(* CoDeSys 2.3.9.50 project: BallGame_template_with_PackMLandDriveFB.pro *)
(* Libraries: TcBase.lib 14.5.09 12:14:08, TcSystem.lib 7.6.16 11:01:22, STANDARD.LIB 5.6.98 12:03:02 *)

(* Task configuration *)
TASK BallGame (PRIORITY := 1, INTERVAL := T#10ms);
	PRG_HMI();
	MAIN();
END_TASK
TASK Drive (PRIORITY := 0, INTERVAL := T#5ms);
	PRG_Drive_Link();
END_TASK

(* Global variable list: Global_Variables *)
VAR_GLOBAL
(* -------------INPUTS and OUTPUTS -------------------*)
(* See Global_Variables_TwinCAT and Global_Variables_CodeSys for
environment specific physical IOs *)

(*-----------------------TIMERS----------------------------*)
	TONMove_Ball_Delay	: TON;
	TONDrive_Delay		: TON;

(*-----------------------COUNTERS----------------------------*)
	CountBallsSortedMetal			: INT:=0;	(*Balls sorted: Metal*)
	CountBallsSortedWooden		: INT:=0;	(*Balls sorted: Wood*)
	CountBallsSortedYellow		: INT:=0;	(*Balls sorted: Wood, Yellow*)
	CountBallsSortedRed			: INT:=0;	(*Balls sorted: Wood, Red*)
	CountBallsSortedBlue			: INT:=0;	(*Balls sorted: Wood, Blue*)
	CountBallsSortedGarbage		: INT:=0;	(*Balls sorted: Unknown*)
	arrCountBallsOnTubes	: ARRAY [1..4] OF INT;	(*Balls on tubes: 1=lower, 2=middle, 3=upper, 4=garbage*)

(*-----------------------FUNCTION BLOCKS----------------*)
	fbDrive				: FB_DriveMovement2;		(*FB for executing the motion*)
	fbStateModel			: FB_StateModel_ST;		(*FB for executing state model*)

(* -------------HMI INPUTS (from HMI to PLC) -------------------*)
	bHMI_BtnStart		: BOOL;		(*Start button on HMI*)

(* -------------HMI OUTPUTS (from PLC to HMI) -------------------*)
	PLC_uModeCurrent	: UINT;		(*Current Mode*)
	PLC_uStateCurrent	: UINT;		(*Current State*)
	O_Light_BeaconRed	: BOOL;		(*Light beacon: Red*)

(*-----------------------OTHER GLOBAL VARS ----------------*)


END_VAR

VAR_GLOBAL CONSTANT
(*-----------------------Lift Position Constants----------------------------*)
	GPOS_LOADING		: WORD := 16#0A;	(*Drive to loading level*)
	GPOS_PIPE_LOW	: WORD := 16#0B;	(*Drive to lower pipe*)
	GPOS_PIPE_MID		: WORD := 16#0C;	(*Drive to middle pipe*)
	GPOS_PIPE_UP		: WORD := 16#0D;	(*Drive to upper pipe*)
	GPOS_GARBAGE		: WORD := 16#0E;	(*Drive to garbage pipe*)
	GPOS_COLOR_SEN	: WORD := 16#0F;	(*Drive to colour sensor*)

(*-----------------------Ball Type Constants----------------------------*)
	METAL				: BOOL := FALSE;
	WOODEN		: BOOL := TRUE;

(*-----------------------TIME Constants----------------------------*)
	T_LOADING_BALL	: TIME := T#1.5s;	(*Delay for ball to roll from Slot2 to Lifter*)
	T_DRIVE_DELAY		: TIME := T#2s;	(*Delay for drive to start movement*)
END_VAR

(* Global variable list: Global_Variables_CodeSys *)
VAR_GLOBAL
(* -------------INPUTS-------------------*)
	ISensorOpt 			:BOOL;	(*Optical sensor - is ball present*)
	ISensorInd 			:BOOL;	(*Inductive sensor - is metal ball present*)
	IEmergencyClear 		:BOOL;	(*Emergency stop is cleared*)
	IRun 				:BOOL;	(*Run switch*)
	ILimitUp 				:BOOL;	(*Lift's limit switch is activated - Up*)
	ILimitLow 		 	:BOOL;	(*Lift's limit switch is activated - Low*)
	IGateClosedMid		:BOOL;	(*Pipe gate closed - Mid*)
	IGateClosedLow		:BOOL;	(*Pipe gate closed - Low*)
	ISorterGateClosed		:BOOL;	(*Sorter gate closed*)
	ISorterLiftUp			:BOOL;	(*Sorter lift at up position*)
	ISorterLiftDown		:BOOL;	(*Sorter lift at down position*)
	IPressureApplied		:BOOL;	(*Pressure is available for the system*)
	TEMP1				:BOOL;
	ISenColourYellow		:BOOL;	(*Colour sensor In1 - Yellow*)
	ISenColourBlue		:BOOL;	(*Colour sensor In2 - Blue*)
	ISenColourGreen		:BOOL;	(*Colour sensor In3 - Green*)
	ISenColourRed		:BOOL;	(*Colour sensor In4 - Red*)
	IDriveStatus 			:WORD;	(*From lift drive status information*)

(* -------------OUTPUTS-------------------*)
	OGateMid			:BOOL;	(*Valve: Open pipe gate - Mid*)
	OGateLow			:BOOL;	(*Valve: Open pipe gate - Low*)
	OSorterGate			:BOOL;	(*Valve: Open sorter gate*)
	OSorterLift			:BOOL;	(*Valve: Sorter lift up*)
	OEjector				:BOOL;	(*Ejector push ball out from lift*)
	ODriveControl 		:WORD;	(*To lift drive control information*)
END_VAR

(* Global variable list: Global_Variables_TwinCAT *)
VAR_GLOBAL
(* -------------INPUTS-------------------*)
	ISensorOpt 		AT %I*	:BOOL;	(*Optical sensor - is ball present*)
	ISensorInd 		AT %I*	:BOOL;	(*Inductive sensor - is metal ball present*)
	IEmergencyClear 	AT %I*	:BOOL;	(*Emergency stop is cleared*)
	IRun 			AT %I*	:BOOL;	(*Run switch*)
	ILimitUp 			AT %I*	:BOOL;	(*Lift's limit switch is activated - Up*)
	ILimitLow 		AT %I* 	:BOOL;	(*Lift's limit switch is activated - Low*)
	IGateClosedMid	AT %I*	:BOOL;	(*Pipe gate closed - Mid*)
	IGateClosedLow	AT %I*	:BOOL;	(*Pipe gate closed - Low*)
	ISorterGateClosed	AT %I*	:BOOL;	(*Sorter gate closed*)
	ISorterLiftUp		AT %I*	:BOOL;	(*Sorter lift at up position*)
	ISorterLiftDown	AT %I*	:BOOL;	(*Sorter lift at down position*)
	IPressureApplied	AT %I*	:BOOL;	(*Pressure is available for the system*)
	TEMP1			AT %I*	:BOOL;
	ISenColourYellow	AT %I*	:BOOL;	(*Colour sensor In1 - Yellow*)
	ISenColourBlue	AT %I*	:BOOL;	(*Colour sensor In2 - Blue*)
	ISenColourGreen	AT %I*	:BOOL;	(*Colour sensor In3 - Green*)
	ISenColourRed	AT %I*	:BOOL;	(*Colour sensor In4 - Red*)
	IDriveStatus 		AT %I*	:WORD;	(*From lift drive status information*)

(* -------------OUTPUTS-------------------*)
	OGateMid		AT %Q*	:BOOL;	(*Valve: Open pipe gate - Mid*)
	OGateLow		AT %Q*	:BOOL;	(*Valve: Open pipe gate - Low*)
	OSorterGate		AT %Q*	:BOOL;	(*Valve: Open sorter gate*)
	OSorterLift		AT %Q*	:BOOL;	(*Valve: Sorter lift up*)
	OEjector			AT %Q*	:BOOL;	(*Ejector push ball out from lift*)
	ODriveControl 	AT %Q*	:WORD;	(*To lift drive control information*)
END_VAR

(* Global variable list: TwinCAT_Configuration *)
(* Generated automatically by TwinCAT - (read only) *)
VAR_CONFIG
	.ISensorOpt AT %IX0.0 : BOOL;	(*  ~ {LinkedWith:TIID^Device 4 (EL6731)^Box 2  (BK3110)^Term 2 (KL1002)^Channel 1^Input} *)
	.ISensorInd AT %IX0.1 : BOOL;	(*  ~ {LinkedWith:TIID^Device 4 (EL6731)^Box 2  (BK3110)^Term 2 (KL1002)^Channel 2^Input} *)
	.IEmergencyClear AT %IX0.2 : BOOL;	(*  ~ {LinkedWith:TIID^Device 4 (EL6731)^Box 2  (BK3110)^Term 3 (KL1002)^Channel 1^Input} *)
	.IRun AT %IX0.3 : BOOL;	(*  ~ {LinkedWith:TIID^Device 4 (EL6731)^Box 2  (BK3110)^Term 3 (KL1002)^Channel 2^Input} *)
	.ILimitUp AT %IX0.4 : BOOL;	(*  ~ {LinkedWith:TIID^Device 4 (EL6731)^Box 2  (BK3110)^Term 4 (KL1002)^Channel 1^Input} *)
	.ILimitLow AT %IX0.5 : BOOL;	(*  ~ {LinkedWith:TIID^Device 4 (EL6731)^Box 2  (BK3110)^Term 4 (KL1002)^Channel 2^Input} *)
	.IGateClosedMid AT %IX0.7 : BOOL;	(*  ~ {LinkedWith:TIID^Device 4 (EL6731)^Box 2  (BK3110)^Term 5 (KL1104)^Channel 2^Input} *)
	.IGateClosedLow AT %IX1.0 : BOOL;	(*  ~ {LinkedWith:TIID^Device 4 (EL6731)^Box 2  (BK3110)^Term 5 (KL1104)^Channel 3^Input} *)
	.ISorterGateClosed AT %IX1.1 : BOOL;	(*  ~ {LinkedWith:TIID^Device 4 (EL6731)^Box 2  (BK3110)^Term 5 (KL1104)^Channel 4^Input} *)
	.ISorterLiftUp AT %IX1.2 : BOOL;	(*  ~ {LinkedWith:TIID^Device 4 (EL6731)^Box 2  (BK3110)^Term 6 (KL1104)^Channel 1^Input} *)
	.ISorterLiftDown AT %IX1.3 : BOOL;	(*  ~ {LinkedWith:TIID^Device 4 (EL6731)^Box 2  (BK3110)^Term 6 (KL1104)^Channel 2^Input} *)
	.IPressureApplied AT %IX1.4 : BOOL;	(*  ~ {LinkedWith:TIID^Device 4 (EL6731)^Box 2  (BK3110)^Term 6 (KL1104)^Channel 3^Input} *)
	.TEMP1 AT %IX1.5 : BOOL;	(*  ~ {LinkedWith:TIID^Device 4 (EL6731)^Box 2  (BK3110)^Term 6 (KL1104)^Channel 4^Input} *)
	.ISenColourYellow AT %IX1.6 : BOOL;	(*  ~ {LinkedWith:TIID^Device 4 (EL6731)^Box 2  (BK3110)^Term 7 (KL1104)^Channel 1^Input} *)
	.ISenColourBlue AT %IX1.7 : BOOL;	(*  ~ {LinkedWith:TIID^Device 4 (EL6731)^Box 2  (BK3110)^Term 7 (KL1104)^Channel 2^Input} *)
	.ISenColourGreen AT %IX2.0 : BOOL;	(*  ~ {LinkedWith:TIID^Device 4 (EL6731)^Box 2  (BK3110)^Term 7 (KL1104)^Channel 3^Input} *)
	.ISenColourRed AT %IX2.1 : BOOL;	(*  ~ {LinkedWith:TIID^Device 4 (EL6731)^Box 2  (BK3110)^Term 7 (KL1104)^Channel 4^Input} *)
	.IDriveStatus AT %IB4 : WORD;	(*  ~ {LinkedWith:TIID^Device 4 (EL6731)^Box 5 (DKC03)^DKC03 mit LSPM2^Inputs^DKC03 mit LSPM2_0_0} *)
	.OGateMid AT %QX0.1 : BOOL;	(*  ~ {LinkedWith:TIID^Device 4 (EL6731)^Box 2  (BK3110)^Term 8 (KL2114)^Channel 2^Output} *)
	.OGateLow AT %QX0.2 : BOOL;	(*  ~ {LinkedWith:TIID^Device 4 (EL6731)^Box 2  (BK3110)^Term 8 (KL2114)^Channel 3^Output} *)
	.OSorterGate AT %QX0.3 : BOOL;	(*  ~ {LinkedWith:TIID^Device 4 (EL6731)^Box 2  (BK3110)^Term 8 (KL2114)^Channel 4^Output} *)
	.OSorterLift AT %QX0.4 : BOOL;	(*  ~ {LinkedWith:TIID^Device 4 (EL6731)^Box 2  (BK3110)^Term 9 (KL2114)^Channel 1^Output} *)
	.OEjector AT %QX0.5 : BOOL;	(*  ~ {LinkedWith:TIID^Device 4 (EL6731)^Box 2  (BK3110)^Term 9 (KL2114)^Channel 2^Output} *)
	.ODriveControl AT %QB2 : WORD;	(*  ~ {LinkedWith:TIID^Device 4 (EL6731)^Box 5 (DKC03)^DKC03 mit LSPM2^Outputs^DKC03 mit LSPM2_1_0} *)
END_VAR

(* Data type *)
TYPE E_ModeCtrl :
(
	eMode_undefined := 0,
	eMode_Automatic :=1,
	eMode_XXX :=2,
	eMode_Manual :=99
);
END_TYPE

(* Data type *)
TYPE E_ModeProc :
(*Procedural control modes. Can be changed in any state*)
(
	eModeProc_undefined := 0,
	eModeProc_Automatic :=1,
	eModeProc_SemiAutomatic :=2,
	eModeProc_Manual :=3
);
END_TYPE

(* Data type *)
TYPE E_State :
(
	eSt_Aborting :=0,
	eSt_Aborted,
	eSt_Clearing,
	eSt_Stopped,
	eSt_Stopping,
	eSt_Resetting,
	eSt_Idle,
	eSt_Starting,
	eSt_Execute,
	eSt_Suspending,
	eSt_Suspended,
	eSt_Unsuspending,
	eSt_Holding,
	eSt_Held,
	eSt_UnHolding,
	eSt_Completing,
	eSt_Completed
);
END_TYPE

(* POU PRG_HMI, ST *)
PROGRAM PRG_HMI
VAR
	(*HMI Buttons*)
	bBtnResetCounters	: BOOL;	(*Button Reset counters*)
	bBtnEmptyPipes		: BOOL;	(*Button Empty Pipes*)

	(*Variables for Lift visualisation*)
	iSorterLiftPos	: INT;		(*Position of Sorter Lift cylinder*)
	iLiftPos		: INT;		(*Position of the lift*)
	wTargetPos	: INT;		(*Current target position of the lift*)
	bBall_InLift	: BOOL;		(*Is there a ball in lift*)

	(*internal variables*)
	RS_Ball_InLift	: RS;		(*Flip-flop for ball in the lift*)
	i: INT := 0;		(*Counter*)
END_VAR
(*Producing blinking signal*)
PRG_Blinking();

(*Sorter lift position calculus*)
IF OSorterLift AND (iSorterLiftPos < 30) THEN
	iSorterLiftPos := iSorterLiftPos +1;
END_IF;
IF NOT OSorterLift AND (iSorterLiftPos > 0) THEN
	iSorterLiftPos := iSorterLiftPos - 1;
END_IF;

(*Lift position calculus*)
CASE fbDrive.wDestination OF
GPOS_PIPE_UP:		(*Go to Pipe Up*)
	wTargetPos:=375;
GPOS_PIPE_MID:	(*Go to Pipe Mid*)
	wTargetPos:=275;
GPOS_COLOR_SEN:	(*Go to Colour sensor*)
	wTargetPos:=220;
GPOS_PIPE_LOW:	(*Go to Pipe Low*)
	wTargetPos:=175;
GPOS_GARBAGE:	(*Go to garbage position*)
	wTargetPos:=110;
GPOS_LOADING:	(*Go to loading position*)
	wTargetPos:=20;
ELSE
	wTargetPos:=0;
END_CASE;

(*Drive lift*)
IF iLiftPos > wTargetPos THEN	(*Lift is higher than target*)
	iLiftPos := iLiftPos - 1;	 (*Go down*)
ELSIF iLiftPos < wTargetPos THEN	(*Lift is lower than target*)
	iLiftPos := iLiftPos + 1;	 (*Go up*)
END_IF;

(*Is there a ball in the lift*)
RS_Ball_InLift(
	SET:= (iLiftPos=20 AND NOT OSorterGate),
	RESET1:=OEjector ,
	Q1=>bBall_InLift );

(* ---------------------------------- Button handlers ---------------------------------- *)
(*Button Empty Pipes*)

(*Button Reset coutners*)
IF bBtnResetCounters THEN
	CountBallsSortedMetal := 0;
	CountBallsSortedWooden := 0;
	CountBallsSortedYellow := 0;
	CountBallsSortedBlue := 0;
	FOR i := 1 TO 3 DO
		arrCountBallsOnTubes[i] := 0;
	END_FOR;
END_IF;
END_PROGRAM

(* POU Programs/PRG_Blinking, ST *)
PROGRAM PRG_Blinking
(*Supporting caluculations: Blinking signals
Author: 	Niko Siltala, niko.siltala@tut.fi
Date: 	2014-01-01*)

VAR_OUTPUT
	bSign4Hz	:BOOL;				(*4 Hz (240krt/min) taajudella vaihteleva signaali*)
	bSign2Hz	:BOOL;				(*2 Hz (120krt/min) taajudella vaihteleva signaali*)
	bSign1Hz	:BOOL;				(*1 Hz (60krt/min) taajudella vaihteleva signaali*)
	bSign0_5Hz	:BOOL;				(*0,5 Hz (30krt/min) taajudella vaihteleva signaali*)
END_VAR
VAR
	bInitDone	: BOOL	:=FALSE;		(*Ohjelman initialisointi*)
	TP_Delay	: TP;					(*Nopein taajuus / 2 tuottaja*)
	bBaseHz	: BOOL	:=FALSE;		(*Nopein taajuus/2*)
	iBaseHz		: UINT	:=4;			(*Base taajuus (Hz)*)
	RTRIG_2Hz_Sign 	: R_TRIG;		(*2Hz signaalin generointi*)
	RTRIG_1Hz_Sign 	: R_TRIG;		(*1Hz signaalin generointi*)
	RTRIG_0_5Hz_Sign	: R_TRIG;	(*0,5Hz signaalin generointi*)
	tBaseTaajuus	:TIME;			(*Base vilkutuksen timerin arvo. f/2*)
	fPLC_CYCLE_TIME	: LREAL;		(*PLC:n cycli aika. Sekunttia*)
END_VAR
(*Ohjelman initialisoinnit - Suoritetaan vain kertaalleen*)
IF NOT bInitDone THEN
	fPLC_CYCLE_TIME := UDINT_TO_LREAL(SystemTaskInfoArr[1].cycleTime) / 10E6;
	(*Base Vilkkusignaalien tuottaminen*)
	(* 250ms - 1* cykliaika(20ms)*)
	tBaseTaajuus := LREAL_TO_TIME( ( (1/ UINT_TO_LREAL(iBaseHz) / 2 ) - 1 * fPLC_CYCLE_TIME ) * 1000);
	bInitDone := TRUE;
END_IF;


(*Base signaalin genrointi*)
TP_Delay(IN:=NOT TP_Delay.Q , PT:=tBaseTaajuus);
IF NOT TP_Delay.Q THEN
	bBaseHz := NOT bBaseHz;
	bSign4Hz:= bBaseHz;
END_IF;

(*2Hz signaalin genrointi*)
RTRIG_2Hz_Sign(CLK:=bSign4Hz);
IF RTRIG_2Hz_Sign.Q THEN
	bSign2Hz:=NOT bSign2Hz;
END_IF;

(*1Hz signaalin genrointi*)
RTRIG_1Hz_Sign(CLK:=bSign2Hz);
IF RTRIG_1Hz_Sign.Q THEN
	bSign1Hz:=NOT bSign1Hz;
END_IF;

(*0,5 Hz signaalin generointi*)
RTRIG_0_5Hz_Sign(CLK:=bSign1Hz);
IF (RTRIG_0_5Hz_Sign.Q) THEN
	bSign0_5Hz:= NOT bSign0_5Hz;
END_IF;
END_PROGRAM

(* POU MAIN, ST *)
PROGRAM MAIN
(*Main program for application. Uses PackML state model to control the execution of the application*)
VAR
	tonStarting			: TON;
END_VAR
(* ****** Section 1: Initialisations and default values. Initial conditions for variables on every PLC cycle*)
(*Default values*)
fbStateModel.bSC := FALSE;

(*System resets*)

(* ****** Section 2: Actions in your program without considering the Control Mode. I.e. actions are performed same way indenpendent on
current Control Mode selection.*)
(*Mode independent state actions. Change / Add / Remove states according your need*)
CASE fbStateModel.eState OF
eSt_Aborting:
	(* One can make specific actions in case of specific Mode-State combination.
	   One can also consider to call a specific program when in specific Mode-State combination*)
	fbStateModel.bSC := TRUE;		(*MODIFY*)
eSt_Clearing:
	fbStateModel.bSC := TRUE;		(*MODIFY*)
eSt_Holding:
	fbStateModel.bSC := TRUE;		(*MODIFY*)
eSt_UnHolding:
	fbStateModel.bSC := TRUE;		(*MODIFY*)
eSt_Suspending:
	fbStateModel.bSC := TRUE;		(*MODIFY*)
eSt_Unsuspending:
	fbStateModel.bSC := TRUE;		(*MODIFY*)
END_CASE;

(* ****** Section 3: Actions in your program which are Control Mode specific. Two nested case structures where outer one selects the
control mode and inner the PackML state. In order to avoid conflicts, it would be better to process each PackML state either in Section 2 
or Section 3, but not in both. *)
(*Execution mode related state actions. Change / Add / Remove mode and states according your need*)
CASE fbStateModel.eMode OF
(*MODE: MANUAL*)
eMode_Manual:
	(* ****** Section 3.1: PackML state based processing actions when Control Mode is Manual.*)
	CASE fbStateModel.eState OF
	eSt_Starting:
		fbStateModel.bSC := TRUE;			(*MODIFY*)
	eSt_Stopping:
		fbStateModel.bSC := TRUE;			(*MODIFY*)
	END_CASE;

(*MODE: AUTOMATIC*)
eMode_Automatic:
	(* ****** Section 3.2: PackML state based processing actions when Control Mode is Automatic.*)
	CASE fbStateModel.eState OF
	eSt_Idle:
		tonStarting(IN:=FALSE , PT:= , Q=> , ET=> );	(*MODIFY*)
	eSt_Starting:
		tonStarting(IN:=TRUE , PT:=T#2s , Q=> , ET=> );	(*MODIFY*)
		fbStateModel.bSC := tonStarting.Q;			(*MODIFY*)
	eSt_Completing:
		fbStateModel.bSC := TRUE;					(*MODIFY*)
	eSt_Completed:
		;
	END_CASE;

(* ****** Section 4: Grouping PackML states for calling Programs or FB instances.
This is to avoid repetition inside above case structure in Section 3. With IF clause setting lower (and upper) state limits we can filter out the states when we want to call 
specific programs. The order of states is defined in Tab:Data types > E_PackMLState. eSt_Aborting is lowest and eSt_Completed is highest.
Here we filter calling programs, only when we are in higher states than Stopped. 
This can be pulled out as completely separated section, like in PackML_StateModel_v2-2.pro project. There is inside IF again CASE which process each Control Mode separately.*)
(*Execution part. Making calls for program if we are on states above Stopped*)
	(*If we are between specific states, make some action or program call*)
	IF  (fbStateModel.eState>eSt_Starting) AND (fbStateModel.eState<=eSt_Completing) THEN
		(*Make here the actions / calls
			Good place to start with is PRG_Sorting (PRG)*)
		; 		(*MODIFY*)
	END_IF;

(*MODE: UNKNOWN*)
ELSE	(*Error*)
	; (*TODO*)
END_CASE;

(* ****** Section 5: Calling the fbStateModel instance.
Here the instance of state model is called and all triggering inputs are set, but bSC (State Completed), which you control in your programs. 
This is indication that your program has  finished certain stage.
- Pay attention where the instance fbStateModel is defined. Do you do it in global variables or e.g. here in PRG_MAIN? Important is to use the 
same instance in all places, so that machine state is unique and shared. Remember, if you have multiple definitions, the PRG_MAIN "hides" 
the global one, and might lead to problems elswhere, when you think you are using the same instance, but actually are not. 
- In case you are using the PackML visualisation (VC_PackMLStates), make sure you connect its placeholder to the very same PackML FB instance.
- The Mask for wIgnoreState is created as following. I use binary base for the value(2#). The lowest bit in the mask corresponds the eSt_Aborting
 in E_PackMLState. The next is eSt_Aborted, and so on. Specific state is ignored and jumped over when it is masked out i.e. ignored by having 1 
in that position. Note that implementation allows this only for selected states. See FB_PackMLStateModel_ST code for further details.*)
(*Calling & Updating the state model*)
(*TODO: Evaluate and change all input conditions according your application needs*)
fbStateModel(
	bResetFB:= ,
	eModeReq:= ,
	wIgnoreState := 2#000000,		(*TODO: Which states should be ignodered. Default: 2#000000 or 2#100000. The latter is ignoring Resetting state*)
	bSC:= ,			(*Must not be assigned ANY variable, because fb input is directly operated!!!*)
	bAbort:= NOT IEmergencyClear,
	bClear:= IEmergencyClear,
	bReset:= ,
	bStart:= IRun,
	bHold:= ,
	bUn_Hold:= ,
	bSuspend:= ,
	bUn_Suspend:= ,
	bStop:= ,
	bComplete:= ,
	bAck_Completed:= ,
	eMode=> PLC_uModeCurrent,
	eState=> PLC_uStateCurrent);

(* ****** Section 6: Here we update all outputs according the current state of our PackML model. This allows us to process the in single location.
The control of outputs is bind to state, not e.g. to inputs. The inputs are the one driving the PackML model forward. Again CASE structure can be used.*)
(*Call for HMI and UI update*)
HMI_and_UI_Update;
END_PROGRAM
ACTION HMI_and_UI_Update:
(*HMI Update*)
PRG_Blinking (bSign4Hz=> , bSign2Hz=> , bSign1Hz=> , bSign0_5Hz=> );
(*Init values*)
O_Light_BeaconRed := FALSE;

(*OLight_Start :=  (fbStateModel.eState >= eSt_Resetting) AND (fbStateModel.eState < eSt_Completed);*)

CASE fbStateModel.eState OF
eSt_Aborting, eSt_Aborted:
	O_Light_BeaconRed := PRG_Blinking.bSign1Hz;
eSt_Clearing:
	O_Light_BeaconRed := PRG_Blinking.bSign0_5Hz;
eSt_Stopped, eSt_Completed:
	O_Light_BeaconRed := TRUE;
eSt_Starting:
	;
END_CASE;
END_ACTION

(* POU Programs/PRG_Drive_Link, FBD *)
PROGRAM PRG_Drive_Link
VAR
END_VAR
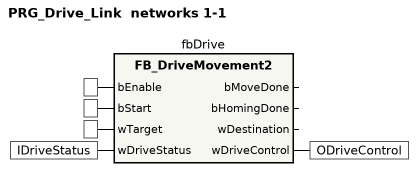
_FBD_ (* Function Block Diagram *)
NETWORK 1
	fbDrive:FB_DriveMovement2(bEnable: , bStart: , wTarget: , wDriveStatus: IDriveStatus, wDriveControl => ODriveControl)
_END_FBD_
END_PROGRAM

(* POU FBs/FB_DriveMovement2, ST *)
FUNCTION_BLOCK FB_DriveMovement2
(* This function block is making all movements for the drive
	bEnable = must be TRUE
	Target = int value of 0 - 63
	bStart = with rising edge starts the movement

	bMoveDone gets true when the movement is finalised.
Author: 	Niko Siltala, niko.siltala@tut.fi
Date: 	2014-01-01*)

VAR_INPUT
	bEnable			: BOOL:=FALSE;	(*Enables the fuction block*)
	bStart			: BOOL:=FALSE;	(*Starts the motion to target by rising edge*)
	wTarget			: WORD:=0;		(*Target destination*)
	wDriveStatus		: WORD;			(*Status word from Indramat Drive*)
END_VAR
VAR_OUTPUT
	bMoveDone		:BOOL:=FALSE;	(*The commanded move has been completed. Drive is at required destination*)
	bHomingDone	:BOOL:=FALSE;	(*Drive has been homed*)
	wDestination		:WORD;			(*Current destination*)
	wDriveControl		:WORD;			(*Control word to Indramat Drive*)
END_VAR
VAR_IN_OUT
END_VAR
VAR
	TONTimer1 	: TON;
	TONTimer2 	: TON;
END_VAR
(*
This function block is making all movements for the drive
	bEnable = must be TRUE
	Target = int value of 0 - 63
	bStart = with rising edge starts the movement

	bMoveDone gets true when the movement is finalised
*)
IF bEnable THEN
	(*Drive is Enabled*)
	wDriveControl:=wDriveControl OR 16#0001;
	IF (wDriveStatus AND 16#0080)>0 AND (wDriveStatus AND 16#0040)>0 THEN
		IF bStart=TRUE THEN
			(*bStart is true*)
			IF bHomingDone=FALSE THEN
				(*Homing procedure*)
				IF TONTimer1.Q=FALSE THEN
					wDriveControl:=16#0005;
					TONTimer1(IN:=TRUE, PT:=T#100ms);(*100ms*)
				ELSE
					IF TONTimer2.Q=FALSE THEN
						(*Start drive*)
						wDriveControl:=16#0007;
						TONTimer2(IN:=TRUE, PT:=T#500ms); (*500ms*)
					ELSE
						(*Timer2 have expired*)
						IF (wDriveStatus AND 16#0004)>0 THEN
							TONTimer1(IN:=FALSE);
							TONTimer2(IN:=FALSE);
							wDriveControl:=16#0001;
							bHomingDone:=TRUE;
						END_IF;
					END_IF;
				END_IF;
			ELSE
				(*Normal movement*)
				IF TONTimer1.Q=FALSE THEN
					(*Set target and Enabled*)
					wDriveControl:=SHL(wTarget,8) OR 16#0001;
					wDestination:=wTarget;
					TONTimer1(IN:=TRUE, PT:=T#10ms);(*10ms*)
				ELSE
					IF TONTimer2.Q=FALSE THEN
						(*Start drive*)
						wDriveControl:=wDriveControl OR 16#0002;
						TONTimer2(IN:=TRUE, PT:=T#500ms); (*500ms*)
					ELSE
						(*Timer2 have expired*)
						IF (wDriveStatus AND 16#0010)>0 THEN
							(*End the movement when user forgets to provide lowering edge*)
							(*bStart:=FALSE;*)
							(*Requested movement is done*)
							bMoveDone:=TRUE;
						END_IF;
					END_IF;
				END_IF; (*Normal movement*)
			END_IF;(*bHomingDone=FALSE*)
		ELSE
			(*bStart is false*)
			bMoveDone:=FALSE;
			TONTimer1(IN:=FALSE);
			TONTimer2(IN:=FALSE);
		END_IF;
	END_IF;
ELSE (*bEnable*)
	(*Drive is NOT Enabled*)
	wDriveControl:=16#0000;
	bMoveDone:=FALSE;
	bHomingDone:=FALSE;
	TONTimer1(IN:=FALSE);
	TONTimer2(IN:=FALSE);
END_IF;
END_FUNCTION_BLOCK

(* POU EXAMPLES, SFC *)
PROGRAM EXAMPLES
VAR
	fbDrive			: DriveMovement2;		(*FB for executing the motion*)
	tonTimer			: TON;			(*Standard TON timer. Use this*)
	fbDelay			: FB_Wait;		(*Different simplified timer.
END_VAR
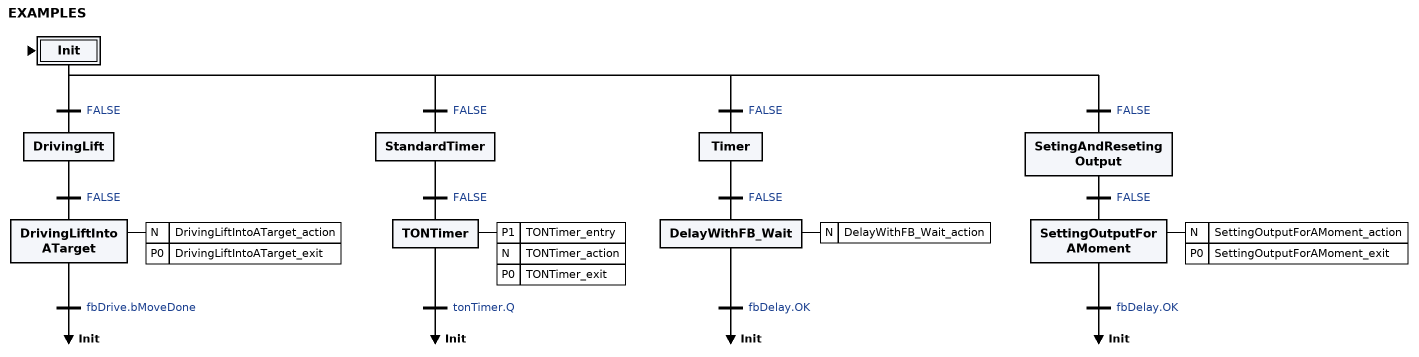
INITIAL_STEP Init:
END_STEP
TRANSITION FROM Init TO DrivingLift := FALSE;
END_TRANSITION
TRANSITION FROM Init TO StandardTimer := FALSE;
END_TRANSITION
TRANSITION FROM Init TO Timer := FALSE;
END_TRANSITION
TRANSITION FROM Init TO SetingAndResetingOutput := FALSE;
END_TRANSITION
STEP DrivingLift:
END_STEP
TRANSITION FROM DrivingLift TO DrivingLiftIntoATarget := FALSE;
END_TRANSITION
STEP DrivingLiftIntoATarget:
	DrivingLiftIntoATarget_action(N);
	DrivingLiftIntoATarget_exit(P0);
END_STEP
TRANSITION FROM DrivingLiftIntoATarget TO Init := fbDrive.bMoveDone;
END_TRANSITION
STEP StandardTimer:
END_STEP
TRANSITION FROM StandardTimer TO TONTimer := FALSE;
END_TRANSITION
STEP TONTimer:
	TONTimer_entry(P1);
	TONTimer_action(N);
	TONTimer_exit(P0);
END_STEP
TRANSITION FROM TONTimer TO Init := tonTimer.Q;
END_TRANSITION
STEP Timer:
END_STEP
TRANSITION FROM Timer TO DelayWithFB_Wait := FALSE;
END_TRANSITION
STEP DelayWithFB_Wait:
	DelayWithFB_Wait_action(N);
END_STEP
TRANSITION FROM DelayWithFB_Wait TO Init := fbDelay.OK;
END_TRANSITION
STEP SetingAndResetingOutput:
END_STEP
TRANSITION FROM SetingAndResetingOutput TO SettingOutputForAMoment := FALSE;
END_TRANSITION
STEP SettingOutputForAMoment:
	SettingOutputForAMoment_action(N);
	SettingOutputForAMoment_exit(P0);
END_STEP
TRANSITION FROM SettingOutputForAMoment TO Init := fbDelay.OK;
END_TRANSITION

ACTION DrivingLiftIntoATarget_action:
(*This executes and drives the lift to desired level (=wTarget)
wTarget is selected from given constants. See:Global Constants*)
fbDrive(
	bEnable:= TRUE,
	bStart:= TRUE,
	wTarget:= GPOS_LOADING);
END_ACTION

ACTION DrivingLiftIntoATarget_exit:
(*Stops the motion*)
fbDrive(
	bStart:= FALSE);
END_ACTION

ACTION TONTimer_entry:
tonTimer(IN:=FALSE);
END_ACTION

ACTION TONTimer_action:
tonTimer(IN:=TRUE , PT:=T#1s, Q=> , ET=> );
END_ACTION

ACTION TONTimer_exit:
tonTimer(IN:=FALSE);
END_ACTION

ACTION DelayWithFB_Wait_action:
(*Timer is counting*)
fbDelay(IN_TIME:=T#1s);
END_ACTION

ACTION SettingOutputForAMoment_action:
(*Timer is counting*)
fbDelay(IN_TIME:=T#500ms);

(*Setting Output*)
OEjector := TRUE;
END_ACTION

ACTION SettingOutputForAMoment_exit:
(*Clearing Output*)
OEjector := FALSE;
END_ACTION
END_PROGRAM

(* POU FBs/FB_Wait, ST *)
FUNCTION_BLOCK FB_Wait
(*Waits the given time and sets output after timer has run till end. When called again timer restarts.
Author: 	Niko Siltala, niko.siltala@tut.fi
Date: 	2014-01-01*)
VAR_INPUT
	IN_TIME	:TIME;		(*Time to wait*)
END_VAR
VAR_OUTPUT
	OK 		: BOOL:=FALSE;	(*Gets true after wait time has expired*)
END_VAR
VAR
	Timer	: TP;
	Falling	: F_TRIG;
END_VAR
IF Timer.Q=TRUE THEN
	(*Call timer block when pulse timer is counting*)
	Timer;
ELSE
	(*Timer has espired. Start it again*)
	Timer(IN:=FALSE);
	Timer(PT:=IN_TIME);
	Timer(IN:=TRUE);
END_IF;
(*Set output. True if timer has expired*)
OK:=NOT Timer.Q;
END_FUNCTION_BLOCK

(* POU Programs/PRG_Initialisation, SFC *)
PROGRAM PRG_Initialisation
(*Template program for system initialisation*)
VAR_INPUT
	bReset		: BOOL := FALSE;	(*Reseting the SFC*)
	bExecute	: BOOL;			(*Executes PRG*)
END_VAR
VAR_OUTPUT
	bDone		: BOOL;		(*Program operations done*)
END_VAR
VAR
(* -------------INTERNAL-------------------*)
	bInitDone		: BOOL:=FALSE;	(*Initialisation done*)


(*System variables. See SFC-flags: http://infosys.beckhoff.com/content/1033/tcplccontrol/html/tcplcctrl_editorsfc.htm?id=24319#SFC-Flags*)
	SFCReset		: BOOL := FALSE;	(*For reseting the SFC*)
END_VAR
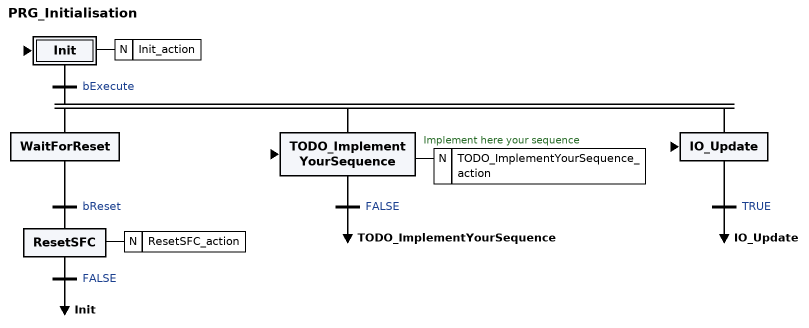
INITIAL_STEP Init:
	Init_action(N);
END_STEP
TRANSITION FROM Init TO (WaitForReset, TODO_ImplementYourSequence, IO_Update) := bExecute;
END_TRANSITION
STEP WaitForReset:
END_STEP
TRANSITION FROM WaitForReset TO ResetSFC := bReset;
END_TRANSITION
STEP TODO_ImplementYourSequence: (* Implement here your sequence *)
	TODO_ImplementYourSequence_action(N);
END_STEP
TRANSITION FROM TODO_ImplementYourSequence TO TODO_ImplementYourSequence := FALSE;
END_TRANSITION
STEP IO_Update:
END_STEP
TRANSITION FROM IO_Update TO IO_Update := TRUE;
END_TRANSITION
STEP ResetSFC:
	ResetSFC_action(N);
END_STEP
TRANSITION FROM ResetSFC TO Init := FALSE;
END_TRANSITION

ACTION Init_action:
(*Clear Reset SFC*)
SFCReset:= FALSE;
END_ACTION

ACTION TODO_ImplementYourSequence_action:
(*Do some actions...

Sulje kaikki portit ... JA tarkista Steppiä seuraavassa transitioehdossa, että kaikki portit ovat kiinni
Close all gates.... and check in following transition that ALL gates are closed*)

;
END_ACTION

ACTION ResetSFC_action:
(*Reset SFC*)
SFCReset:=TRUE;
END_ACTION
END_PROGRAM

(* POU Programs/PRG_Sorting, SFC *)
PROGRAM PRG_Sorting
(*Template program for sorting operation*)
VAR_INPUT
	bReset		: BOOL := FALSE;	(*Reseting the SFC*)
	bExecute	: BOOL;			(*Executes PRG*)
END_VAR
VAR_OUTPUT
	bDone		: BOOL;		(*Program operations done*)
END_VAR
VAR
(* -------------INTERNAL-------------------*)
	bInitDone		: BOOL:=FALSE;	(*Initialisation done*)


(*System variables. See SFC-flags: http://infosys.beckhoff.com/content/1033/tcplccontrol/html/tcplcctrl_editorsfc.htm?id=24319#SFC-Flags*)
	SFCReset		: BOOL := FALSE;	(*For reseting the SFC*)
END_VAR
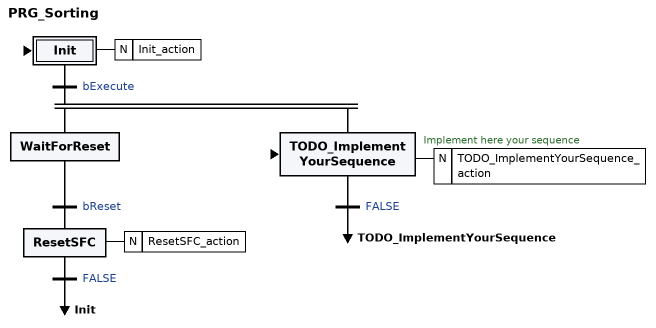
INITIAL_STEP Init:
	Init_action(N);
END_STEP
TRANSITION FROM Init TO (WaitForReset, TODO_ImplementYourSequence) := bExecute;
END_TRANSITION
STEP WaitForReset:
END_STEP
TRANSITION FROM WaitForReset TO ResetSFC := bReset;
END_TRANSITION
STEP TODO_ImplementYourSequence: (* Implement here your sequence *)
	TODO_ImplementYourSequence_action(N);
END_STEP
TRANSITION FROM TODO_ImplementYourSequence TO TODO_ImplementYourSequence := FALSE;
END_TRANSITION
STEP ResetSFC:
	ResetSFC_action(N);
END_STEP
TRANSITION FROM ResetSFC TO Init := FALSE;
END_TRANSITION

ACTION Init_action:
(*Clear Reset SFC*)
SFCReset:= FALSE;
END_ACTION

ACTION TODO_ImplementYourSequence_action:
(*Do some actions...

Sulje kaikki portit ... JA tarkista Steppiä seuraavassa transitioehdossa, että kaikki portit ovat kiinni
Close all gates.... and check in following transition that ALL gates are closed*)

;
END_ACTION

ACTION ResetSFC_action:
(*Reset SFC*)
SFCReset:=TRUE;
END_ACTION
END_PROGRAM

(* POU FBs/FB_StateModel_ST, ST *)
FUNCTION_BLOCK FB_StateModel_ST
(*PackML State model implementation. Slightly modified implementation.
Author: 	Niko Siltala, niko.siltala@tut.fi
Date: 	2016-01-29
*)
VAR_INPUT
	bResetFB	: BOOL;		(*Resets whole FB*)
	eModeReq	: E_ModeCtrl;	(*Requested mode*)
	wIgnoreState	: DWORD;	(*Ignoring states. See bit from E_State definition. Aborting = bit0*)
	bSC			: BOOL;		(*Step Completed acknoledgement*)
	bAbort		: BOOL;		(*Abortting signal = EmergencyStop*)
	bClear		: BOOL;		(*Clear signal*)
	bReset		: BOOL;		(*Reseting signal*)
	bStart		: BOOL;		(*Start signal*)
	bHold		: BOOL;		(*Hold signal*)
	bUn_Hold	: BOOL;		(*Un-Hold signal*)
	bSuspend	: BOOL;		(*Suspend signal*)
	bUn_Suspend	: BOOL;		(*Un-Suspend signal*)
	bStop		: BOOL;		(*Stop signal*)
	bComplete	: BOOL;		(*Complete signal*)
	bAck_Completed	: BOOL;	(*Acknoledgement for Complete signal*)
END_VAR
VAR_OUTPUT
	eMode	: E_ModeCtrl;	(*Current mode*)
	eState	: E_State;	(*Current state*)
END_VAR
VAR
	RTrig_bSC	: R_TRIG; 	(*Rising trigger for State Completed*)
	RTrig_StateChange	: R_TRIG; 	(*Rising trigger for State signal*)
	bResetLocal		: BOOL:=FALSE;	(*Paikallinen Reset*)
	bInitDone	: BOOL;		(*Initialisation*)
END_VAR
IF bResetFB THEN	(*Reseting FB*)
	bInitDone := FALSE;
END_IF;

(*Initialisation*)
IF NOT bInitDone THEN
	eState:= eSt_Aborting;
	bInitDone:=TRUE;
END_IF;

(*Rising triggers monitor*)
RTrig_bSC(CLK:=bSC , Q=> );

(*Abort signal interrupt*)
IF bAbort AND (eState > eSt_Clearing) THEN
	eState:=eSt_Aborting;
END_IF;

(*Stop signal interrupt*)
IF bStop AND (eState > eSt_Stopping) THEN
	eState:=eSt_Stopping;
END_IF;


(*Main case structure*)
CASE eState OF
eSt_Aborting:
	IF bSC THEN
		eState:=eSt_Aborted;
	END_IF;

eSt_Aborted:
	eMode:=eModeReq;	(*Change Mode*)
	IF bClear AND NOT bAbort THEN
		eState:=eSt_Clearing;
	END_IF;

eSt_Clearing:
	IF bAbort THEN
		eState:=eSt_Aborting;
	ELSIF bSC THEN
		eState:=eSt_Stopped;
		RTrig_StateChange(CLK:=bReset , Q=> );
	END_IF;

eSt_Stopping:
	IF bSC THEN
		eState:=eSt_Stopped;
		RTrig_StateChange(CLK:=bReset , Q=> );
	END_IF;

eSt_Stopped:
	eMode:=eModeReq;	(*Change Mode*)
	RTrig_StateChange(CLK:=bReset , Q=> );
(*	ELSIF NOT bStop AND (RTrig_StateChange.Q OR (wIgnoreState.5 AND bStart) ) THEN*)
	IF NOT bStop THEN	(*Stop signal is not active.*)
		IF wIgnoreState.5 AND bStart THEN	(*Reset state is ignored and going directly to start *)
			eState:=eSt_Idle;
		ELSIF RTrig_StateChange.Q THEN 	(*Rising edge for reset*)
			eState:=eSt_Resetting;
		END_IF;
	END_IF;

eSt_Resetting:
	IF bSC OR wIgnoreState.5 THEN
		eState:=eSt_Idle;
	END_IF;

eSt_Idle:
	eMode:=eModeReq;	(*Change Mode*)
	IF bStart OR wIgnoreState.6 THEN
		eState:=eSt_Starting;
	END_IF;

eSt_Starting:
	IF bSC OR wIgnoreState.7 THEN
		eState:=eSt_Execute;
	END_IF;

eSt_Execute:
	IF bComplete THEN
		eState:=eSt_Completing;
	ELSIF bHold THEN
		eState:=eSt_Holding;
	ELSIF bSuspend THEN
		eState:=eSt_Suspending;
	END_IF;

eSt_Holding:
	IF bSC THEN
		eState:=eSt_Held;
	END_IF;

eSt_Held:
	IF bUn_Hold AND NOT bHold THEN
		eState:=eSt_UnHolding;
	END_IF;

eSt_UnHolding:
	IF bSC THEN
		eState:=eSt_Execute;
	END_IF;

eSt_Suspending:
	IF bSC THEN
		eState:=eSt_Suspended;
	END_IF;

eSt_Suspended:
	IF bUn_Suspend AND NOT bSuspend THEN
		eState:=eSt_Unsuspending;
	END_IF;

eSt_Unsuspending:
	IF bSC THEN
		eState:=eSt_Execute;
	END_IF;

eSt_Completing:
	IF RTrig_bSC.Q THEN
		eState:=eSt_Completed;
	END_IF;

eSt_Completed:
	IF bAck_Completed THEN
		eState:=eSt_Resetting;
	END_IF;

ELSE
	(*Default error handler. Undefined state set*)
	eState:=eSt_Aborting;
END_CASE;
END_FUNCTION_BLOCK

(* Visualisation FBs_Visu/FB_DriveMovement2
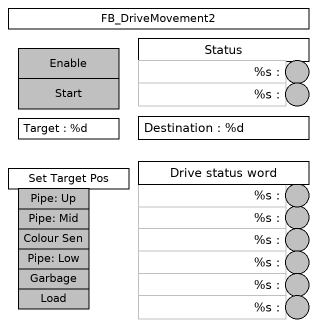
rectangle at (0,0)-(301,21): text "FB_DriveMovement2"
embedded screen at (130,30)-(301,311): FB_VC_Drive_Status
rectangle at (10,110)-(111,131): text "Target : %d"; shows $FB$.wTarget
rectangle at (10,40)-(111,71): text "Enable"; alarm colour if $FB$.bEnable; toggles $FB$.bEnable
rectangle at (10,70)-(111,101): text "Start"; alarm colour if $FB$.bStart; toggles $FB$.bStart
rectangle at (10,280)-(81,301): text "Load"; alarm colour if $FB$.wTarget = .GPOS_LOADING; runs INTERN ASSIGN $FB$.wTarget:=(GPOS_LOADING)
rectangle at (10,260)-(81,281): text "Garbage"; alarm colour if $FB$.wTarget = .GPOS_GARBAGE; runs INTERN ASSIGN $FB$.wTarget:=(GPOS_GARBAGE)
rectangle at (0,160)-(121,181): text "Set Target Pos"
rectangle at (10,240)-(81,261): text "Pipe: Low"; alarm colour if $FB$.wTarget = .GPOS_PIPE_LOW; runs INTERN ASSIGN $FB$.wTarget:=(GPOS_PIPE_LOW)
rectangle at (10,220)-(81,241): text "Colour Sen"; alarm colour if $FB$.wTarget = .GPOS_COLOR_SEN; runs INTERN ASSIGN $FB$.wTarget:=(GPOS_COLOR_SEN)
rectangle at (10,200)-(81,221): text "Pipe: Mid"; alarm colour if $FB$.wTarget = .GPOS_PIPE_MID; runs INTERN ASSIGN $FB$.wTarget:=(GPOS_PIPE_MID)
rectangle at (10,180)-(81,201): text "Pipe: Up"; alarm colour if $FB$.wTarget = .GPOS_PIPE_UP; runs INTERN ASSIGN $FB$.wTarget:=(GPOS_PIPE_UP)
1 more shapes without text or variables
*)

(* Visualisation FBs_Visu/FB_VC_Drive_Status
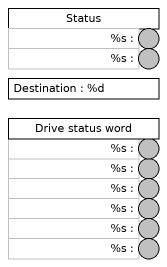
embedded screen at (0,150)-(151,171): VC_BOOLEANSTATUS
rectangle at (0,0)-(151,21): text "Status"
embedded screen at (0,170)-(151,191): VC_BOOLEANSTATUS
embedded screen at (0,130)-(151,151): VC_BOOLEANSTATUS
embedded screen at (0,190)-(151,211): VC_BOOLEANSTATUS
embedded screen at (0,210)-(151,231): VC_BOOLEANSTATUS
embedded screen at (0,230)-(151,251): VC_BOOLEANSTATUS
rectangle at (0,70)-(151,91): text "Destination : %d"; shows $FB$.wDestination
rectangle at (0,110)-(151,131): text "Drive status word"
embedded screen at (0,20)-(151,41): VC_BOOLEANSTATUS
embedded screen at (0,40)-(151,61): VC_BOOLEANSTATUS
*)

(* Visualisation V_Drive
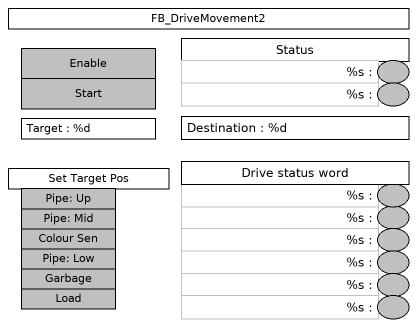
embedded screen at (0,0)-(401,311): FB_DriveMovement2
*)

(* Visualisation V_MAIN
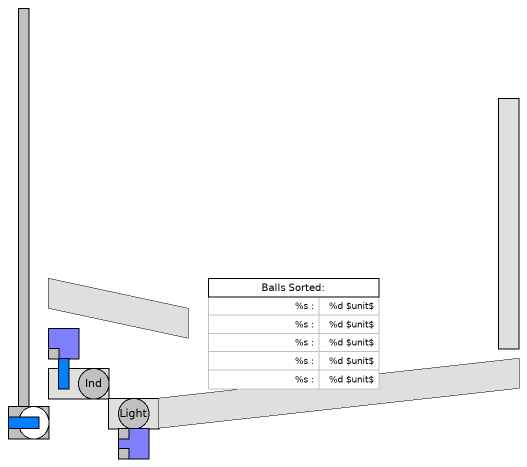
embedded screen at (60,320)-(531,451): VC_Graph_Sorter
embedded screen at (20,0)-(61,431): VC_Graph_Lift
embedded screen at (220,270)-(391,381): VC_Graph_Counters
2 more shapes without text or variables
*)

(* Visualisation Components/VC_BOOLEANSTATUS
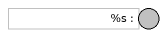
rectangle at (0,0)-(131,21): text "%s :"; shows $Name$
ellipse at (130,0)-(151,21): alarm colour if $bFlag$
*)

(* Visualisation Components/VC_Graph_Counters
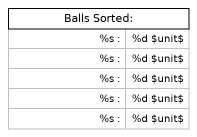
embedded screen at (0,20)-(181,41): VC_Var_Int
rectangle at (0,0)-(181,21): text "Balls Sorted:"
embedded screen at (0,40)-(181,61): VC_Var_Int
embedded screen at (0,60)-(181,81): VC_Var_Int
embedded screen at (0,80)-(181,101): VC_Var_Int
embedded screen at (0,100)-(181,121): VC_Var_Int
*)

(* Visualisation Components/VC_GRAPH_LIFT
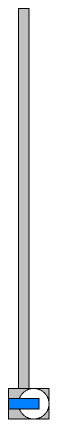
rectangle at (0,380)-(41,411): y offset -1 * PRG_HMI.iLiftPos
ellipse at (10,380)-(41,411): invisible if NOT .PRG_HMI.bBall_InLift; y offset -1 * PRG_HMI.iLiftPos
rectangle at (0,390)-(31,401): invisible if NOT .OEjector; y offset -1 * PRG_HMI.iLiftPos
1 more shapes without text or variables
*)

(* Visualisation Components/VC_GRAPH_SORTER
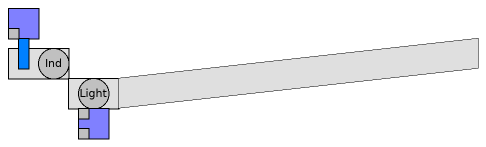
rectangle at (60,70)-(111,101): y offset -1 * PRG_HMI.iSorterLiftPos
rectangle at (10,30)-(21,61): invisible if .OSorterGate
ellipse at (70,70)-(101,101): text "Light"; alarm colour if .ISensorOpt; y offset -1 * PRG_HMI.iSorterLiftPos
ellipse at (30,40)-(61,71): text "Ind"; alarm colour if .ISensorInd
rectangle at (70,100)-(81,111): alarm colour if .ISorterLiftUp
rectangle at (70,120)-(81,131): alarm colour if .ISorterLiftDown
rectangle at (0,20)-(11,31): alarm colour if .ISorterGateClosed
6 more shapes without text or variables
*)

(* Visualisation Visual Components/VC_PackMLStates
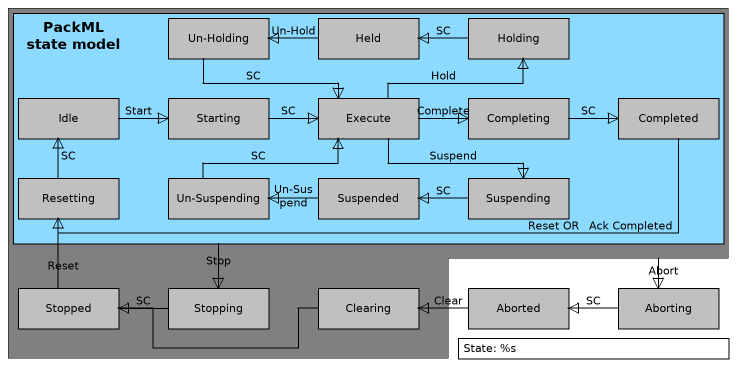
rounded rectangle at (160,280)-(261,321): text "Stopping"; alarm colour if $PackML$.eState = 4
rounded rectangle at (10,90)-(111,131): text "Idle"; alarm colour if $PackML$.eState = 6
rounded rectangle at (160,170)-(261,211): text "Un-Suspending"; alarm colour if $PackML$.eState = 11
rounded rectangle at (610,280)-(711,321): text "Aborting"; alarm colour if $PackML$.eState = 0
rounded rectangle at (460,280)-(561,321): text "Aborted"; alarm colour if $PackML$.eState = 1
rectangle at (450,330)-(721,351): text "State: %s"; shows $PackML$.strState
rounded rectangle at (310,280)-(411,321): text "Clearing"; alarm colour if $PackML$.eState = 2
rounded rectangle at (10,280)-(111,321): text "Stopped"; alarm colour if $PackML$.eState = 3
rounded rectangle at (10,170)-(111,211): text "Resetting"; alarm colour if $PackML$.eState = 5
rounded rectangle at (160,90)-(261,131): text "Starting"; alarm colour if $PackML$.eState = 7
rounded rectangle at (310,90)-(411,131): text "Execute"; alarm colour if $PackML$.eState = 8
rounded rectangle at (460,90)-(561,131): text "Completing"; alarm colour if $PackML$.eState = 15
rounded rectangle at (610,90)-(711,131): text "Completed"; alarm colour if $PackML$.eState = 16
rounded rectangle at (310,170)-(411,211): text "Suspended"; alarm colour if $PackML$.eState = 10
rounded rectangle at (460,170)-(561,211): text "Suspending"; alarm colour if $PackML$.eState = 9
rounded rectangle at (460,10)-(561,51): text "Holding"; alarm colour if $PackML$.eState = 12
rounded rectangle at (310,10)-(411,51): text "Held"; alarm colour if $PackML$.eState = 13
rounded rectangle at (160,10)-(261,51): text "Un-Holding"; alarm colour if $PackML$.eState = 14
polyline at (645,250)-(655,280): alarm colour if $PackML$.bAbort
rectangle at (635,255)-(676,271): text "Abort"; alarm colour if $PackML$.bAbort
polyline at (205,235)-(215,280): alarm colour if $PackML$.bStop
rectangle at (190,245)-(231,261): text "Stop"; alarm colour if $PackML$.bStop
polyline at (195,130)-(335,170): alarm colour if $PackML$.bSC
rectangle at (235,140)-(266,156): text "SC"; alarm colour if $PackML$.bSC
polyline at (195,50)-(335,90): alarm colour if $PackML$.bSC
polyline at (380,50)-(520,90): alarm colour if $PackML$.bHold
rectangle at (420,60)-(451,76): text "Hold"; alarm colour if $PackML$.bHold
polyline at (560,295)-(610,305): alarm colour if $PackML$.bSC
polyline at (45,210)-(55,280): alarm colour if $PackML$.bReset
polyline at (110,105)-(160,115): alarm colour if $PackML$.bStart
polyline at (110,295)-(310,340): alarm colour if $PackML$.bSC
rectangle at (230,60)-(261,76): text "SC"; alarm colour if $PackML$.bSC
polyline at (380,130)-(520,170): alarm colour if $PackML$.bSuspend
rectangle at (415,140)-(476,156): text "Suspend"; alarm colour if $PackML$.bSuspend
rectangle at (120,285)-(151,301): text "SC"; alarm colour if $PackML$.bSC
rectangle at (570,285)-(601,301): text "SC"; alarm colour if $PackML$.bSC
polyline at (410,295)-(460,305): alarm colour if $PackML$.bClear
rectangle at (420,285)-(461,301): text "Clear"; alarm colour if $PackML$.bClear
polyline at (260,105)-(310,115): alarm colour if $PackML$.bSC
rectangle at (265,95)-(296,111): text "SC"; alarm colour if $PackML$.bSC
rectangle at (110,95)-(151,111): text "Start"; alarm colour if $PackML$.bStart
rectangle at (35,250)-(76,266): text "Reset"; alarm colour if $PackML$.bReset
polyline at (410,185)-(460,195): alarm colour if $PackML$.bSC
rectangle at (420,175)-(451,191): text "SC"; alarm colour if $PackML$.bSC
polyline at (410,25)-(460,35): alarm colour if $PackML$.bSC
rectangle at (420,15)-(451,31): text "SC"; alarm colour if $PackML$.bSC
polyline at (260,185)-(310,195): alarm colour if $PackML$.bUn_Suspend
rectangle at (260,170)-(311,206): text "Un-Sus / pend"; alarm colour if $PackML$.bUn_Suspend
polyline at (260,25)-(310,35): alarm colour if $PackML$.bUn_Hold
rectangle at (260,15)-(311,31): text "Un-Hold"; alarm colour if $PackML$.bUn_Hold
polyline at (410,105)-(460,115): alarm colour if $PackML$.bComplete
rectangle at (410,95)-(461,111): text "Complete"; alarm colour if $PackML$.bComplete
polyline at (560,105)-(610,115): alarm colour if $PackML$.bSC
rectangle at (565,95)-(596,111): text "SC"; alarm colour if $PackML$.bSC
polyline at (45,130)-(55,170): alarm colour if $PackML$.bSC
rectangle at (45,140)-(76,156): text "SC"; alarm colour if $PackML$.bSC
polyline at (50,130)-(670,225): alarm colour if $PackML$.bReset OR $PackML$.Ack_Completed
rectangle at (515,210)-(576,226): text "Reset OR"; alarm colour if $PackML$.bReset
rectangle at (575,210)-(671,226): text "Ack Completed"; alarm colour if $PackML$.bAck_Completed
rectangle at (10,10)-(121,51): text "PackML / state model"
2 more shapes without text or variables
*)

(* Visualisation Components/VC_Var_Int
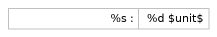
rectangle at (0,0)-(131,21): text "%s :"; shows $Name$
rectangle at (130,0)-(201,21): text "%d $unit$"; shows $VAR$
*)
